(* CoDeSys 2.3 export: INTER_EVENT.EXP *)

(* POU INTER_EVENT, ST *)
FUNCTION_BLOCK INTER_EVENT
VAR_INPUT
	IN: BOOL;
END_VAR
VAR_OUTPUT
	ON: BOOL;
	OFF: BOOL;
END_VAR
VAR
	MTRIG: R_TRIG;
	DTRIG: F_TRIG;
END_VAR
(* Get the ON or OFF event on an input *)

MTRIG(CLK := IN);
ON := MTRIG.Q;
DTRIG(CLK := IN);
OFF := DTRIG.Q;
END_FUNCTION_BLOCK
